FUNCTION_BLOCK POU_1
VAR_INPUT
END_VAR
VAR_OUTPUT
END_VAR
VAR
	TOF_0: TOF;
END_VAR

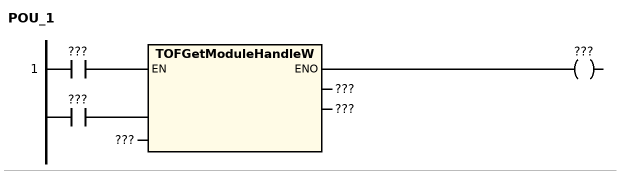
// NETWORK 1
TOFGetModuleHandleW(???, ???);
??? := TRUE;

END_FUNCTION_BLOCK

(* stored: Version 1.1.0.1, ProductVersion 3.1.4024.11
   POU POU_1: Id {54b2a554-2ad8-0499-1755-3aba33758dad}, SpecialFunc None *)
